// TIA Portal V19 export
DATA_BLOCK "DB_PNOZ_Send"   // DB363
{ S7_Optimized_Access := 'FALSE' }
// stored: AutoNumber false
   VAR
      Out : Struct
         Header : Array[0..7] of Byte;
         VirtualOutput : Array[0..127] of Bool;
         LED : Byte;
         Req_Table_Nr : Byte;   // Table Nr
         Segment : Struct
            Req_Nr : Byte;
            Byte_0 : Byte;
            Byte_1 : Byte;
            Byte_2 : Byte;
            Byte_3 : Byte;
            Byte_4 : Byte;
            Byte_5 : Byte;
            Byte_6 : Byte;
            Byte_7 : Byte;
            Byte_8 : Byte;
            Byte_9 : Byte;
            Byte_10 : Byte;
            Byte_11 : Byte;
            Byte_12 : Byte;
         END_STRUCT;
         reserviert : Byte;
         Checksum : Byte := BYTE#16#A4;   // Checksumme, Byte 4 + Byte 39
         Endekennung : Byte := BYTE#16#10;   // last Byte, must be 0x10 every time!
         Struct_Auffueller : Byte;
      END_STRUCT;
   END_VAR
BEGIN
   Out.Header[0] := BYTE#16#05;
   Out.Header[1] := BYTE#16#15;
   Out.Header[3] := BYTE#16#26;
   Out.Header[4] := BYTE#16#5C;
END_DATA_BLOCK
